FUNCTION_BLOCK ProcessState
VAR_INPUT
END_VAR
VAR_OUTPUT
END_VAR
VAR
	m_values: ARRAY [ResiConst.ARR_MIN..ResiConst.STATE_ARR_MAX] OF SValue;
	m_ptrRaConnector: POINTER TO RaConnector;
	
	m_varExp: ValueExpression(EDataType.numeric, FALSE, 0, '', TRUE);
END_VAR

// manages all the system variables

METHOD ProvideServices : BOOL
VAR_INPUT
	i_ptrRaConnector: POINTER TO RaConnector;
END_VAR
m_ptrRaConnector := i_ptrRaConnector;
END_METHOD

METHOD Retrieve : SValue
VAR_INPUT
	i_id: UINT;
	i_checkDef: BOOL;
END_VAR
VAR
	m_val: SValue;
END_VAR
m_val := m_values[i_id];

IF i_checkDef THEN
	IF m_val.Defined THEN
		Retrieve:= m_val;
	ELSE
		m_varExp.FB_init(FALSE, FALSE, EDataType.numeric, FALSE, i_id, '', TRUE);
		m_ptrRaConnector^.RequestRecovery(m_varExp, 'ProcessState.Retrieve');
	END_IF	
ELSE
	Retrieve := m_val;
END_IF
END_METHOD

METHOD SetValue : BOOL
VAR_INPUT
	i_id: UINT;
	i_val: SValue;
END_VAR
SetValue := FALSE;
m_values[i_id].DataType := i_val.DataType;
m_values[i_id].Defined := i_val.Defined;

CASE i_val.DataType OF
	EDataType.binary:
		m_values[i_id].Value.Binary := i_val.Value.Binary;
		SetValue := TRUE;
		
	EDataType.numeric:
		m_values[i_id].Value.Numeric := i_val.Value.Numeric;
		SetValue := TRUE;
		
	EDataType.string_t:
		m_values[i_id].Value.String_t := i_val.Value.String_t;
		SetValue := TRUE;
END_CASE
END_METHOD

METHOD UpdateState_Binary : BOOL
VAR_INPUT
	i_id: UINT;
	i_value: BOOL;
	
	// writes even if the existing data type does not match
	i_force: BOOL;
END_VAR
IF i_force THEN
	m_values[i_id].DataType := EDataType.binary;
	m_values[i_id].Value.Binary := FALSE;
END_IF

IF m_values[i_id].DataType = EDataType.binary THEN
	m_values[i_id].Value.Binary := i_value;
	UpdateState_Binary := TRUE;
ELSE
	UpdateState_Binary := FALSE;
END_IF
END_METHOD

METHOD UpdateState_Defined : BOOL
VAR_INPUT
	i_id: UINT;
	i_defined: BOOL;
END_VAR
m_values[i_id].Defined := i_defined;
UpdateState_Defined := TRUE;
END_METHOD

METHOD UpdateState_Numeric : BOOL
VAR_INPUT
	i_id: UINT;
	i_value: LREAL;
	
	// writes even if the existing data type does not match
	i_force: BOOL;
END_VAR
IF i_force THEN
	m_values[i_id].DataType := EDataType.numeric;
	m_values[i_id].Value.Numeric := 0;
END_IF

IF m_values[i_id].DataType = EDataType.numeric THEN
	m_values[i_id].Value.Numeric := i_value;
	UpdateState_Numeric := TRUE;
ELSE
	UpdateState_Numeric := FALSE;
END_IF
END_METHOD

METHOD UpdateState_NumericIncrement : BOOL
VAR_INPUT
	i_id: UINT;
	
	// writes even if the existing data type does not match
	i_force: BOOL;
END_VAR
IF i_force THEN
	m_values[i_id].DataType := EDataType.numeric;
END_IF

IF m_values[i_id].DataType = EDataType.numeric THEN
	m_values[i_id].Value.Numeric := m_values[i_id].Value.Numeric + 1;
	UpdateState_NumericIncrement := TRUE;
ELSE
	UpdateState_NumericIncrement := FALSE;
END_IF
END_METHOD

METHOD UpdateState_String : BOOL
VAR_INPUT
	i_id: UINT;
	i_value: STRING;
	
	// writes even if the existing data type does not match
	i_force: BOOL;
END_VAR
IF i_force THEN
	m_values[i_id].DataType := EDataType.string_t;
	m_values[i_id].Value.String_t := '';
END_IF

IF m_values[i_id].DataType = EDataType.string_t THEN
	m_values[i_id].Value.String_t := i_value;
	UpdateState_String := TRUE;
ELSE
	UpdateState_String := FALSE;
END_IF
END_METHOD

END_FUNCTION_BLOCK

(* stored: Version 1.1.0.1, ProductVersion 3.1.4024.12
   POU ProcessState: Id {ec18b207-8211-4814-8766-e09236d87b7a}, SpecialFunc None
   Method ProvideServices: Id {c05109a8-c70a-45aa-8b3b-b721a0b3b5a1}
   Method Retrieve: Id {0e3dcca9-10f6-48c6-bcec-257b624314af}
   Method SetValue: Id {1f66cedc-63f4-4624-a6f2-3ae03a91a9b0}
   Method UpdateState_Binary: Id {f24f9c25-e30c-4e3b-81cd-9abfc8d9bb8c}
   Method UpdateState_Defined: Id {8cdc22d2-b29e-44a4-a651-6138a603d0e0}
   Method UpdateState_Numeric: Id {d1b3db2a-e951-4b51-8ff5-aebf8bc96701}
   Method UpdateState_NumericIncrement: Id {1cfa2e4f-a1f3-46ec-91f7-e0243d4728c1}
   Method UpdateState_String: Id {681ea6d1-a1df-47b0-add3-adfe550f3002} *)
